FUNCTION_BLOCK PICKER_HMI_PROXY_NEW (* Communication Unit for HMI using a plug *)
  (* Standard: 61499-2 *)
  (* Version 0.2, 2003-12-05, JHC, Rockwell Automation, Renamed from NEWCOMPFB. *)
  (* Version 0.1, 2002-01-08, JHC, Rockwell Automation, Added DLY FB as example. *)
  (* Version 0.0, 2000-05-27, JHC, Rockwell Automation *)
  (* Compiler header: package fb.rt.pnp;import fb.rt.net.*; *)
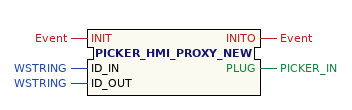
  EVENT_INPUT
    INIT; (* Initialization Request *)
  END_EVENT
  EVENT_OUTPUT
    INITO; (* Initialization Confirm *)
  END_EVENT
  VAR_INPUT
    ID_IN : WSTRING;
    ID_OUT : WSTRING;
  END_VAR
  PLUGS
    PLUG : PICKER_IN;
  END_PLUGS
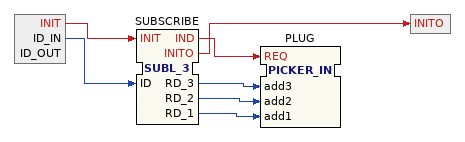
  FBS
    SUBSCRIBE : SUBL_3;
  END_FBS
  EVENT_CONNECTIONS
    SUBSCRIBE.IND TO PLUG.REQ;
    INIT TO SUBSCRIBE.INIT;
    SUBSCRIBE.INITO TO INITO;
  END_CONNECTIONS
  DATA_CONNECTIONS
    ID_IN TO SUBSCRIBE.ID;
    SUBSCRIBE.RD_3 TO PLUG.add3;
    SUBSCRIBE.RD_2 TO PLUG.add2;
    SUBSCRIBE.RD_1 TO PLUG.add1;
  END_CONNECTIONS
END_FUNCTION_BLOCK
